FUNCTION INTERNAL _RegisterComponent : Result
VAR_INPUT
    iComponent  : I_Component;
END_VAR

// Check if the runtime system has been initialized
IF NOT _Runtime.bInit THEN
    // If not initialized, return with an initialization error
    _RegisterComponent := Err.Init;
    RETURN;
END_IF

// Validate that there is an entity currently under construction and the component reference is valid
IF _Ec.iUnderConstruction = 0 OR iComponent = 0 THEN
    // If either is invalid, return interface error
    _RegisterComponent := Err.Itf0;
    RETURN;
END_IF

// Ensure the entity under construction is in the 'Registered' state
IF _Ec.iUnderConstruction._State <> _EntityState.Registered THEN
    // If not registered, the entity context is invalid for component registration
    _RegisterComponent := Err.NotFound;
    RETURN;
END_IF

// Ensure the component is not already assigned to another entity
IF iComponent._Entity <> 0 THEN
    // Component is already linked to an entity, return incorrect argument error
    _RegisterComponent := Err.IncArg;
    RETURN;
END_IF

// Add entity as parent
iComponent._Entity := _Ec.iUnderConstruction._AsIEntity;
iComponent._Entity._Size := iComponent._Entity._Size + 1;

// If the entity already has components, append this one to the end of the component list
IF _Ec.iUnderConstruction._LastComp <> 0 THEN
    _Ec.iUnderConstruction._LastComp._Next := iComponent;           // Link previous last to new component
    iComponent._Prev := _Ec.iUnderConstruction._LastComp;           // Link new component back to previous last
    _Ec.iUnderConstruction._LastComp := iComponent;                 // Update the last component pointer
    _RegisterComponent := Ok;

// If this is the first component being added, initialize the list
ELSE
    _Ec.iUnderConstruction._FirstComp := iComponent;                // Set as first component
    _Ec.iUnderConstruction._LastComp := iComponent;                 // Also set as last component
    _RegisterComponent := Ok;
END_IF

END_FUNCTION

(* stored: Version 1.1.0.1
   POU _RegisterComponent: Id {c4cd3965-1528-4d1c-ab1a-c99e9a28aeba}, SpecialFunc None *)
